// TwinCAT 3 PLC project MC
// ProgramVersion: 3.1.4024.0
// libraries:
//   Tc2_Math, * (Beckhoff Automation GmbH)
//   Tc2_MC2, * (Beckhoff Automation GmbH)
//   Tc2_Standard, * (Beckhoff Automation GmbH)
//   Tc2_System, * (Beckhoff Automation GmbH)
//   Tc2_Utilities, * (Beckhoff Automation GmbH)
//   Tc3_MC2_AdvancedHoming, * (Beckhoff Automation GmbH)
//   Tc3_Module, * (Beckhoff Automation GmbH)
// project tree:
//   GVLs/ motor_settings.TcGVL, robot_settings.TcGVL
//   / PlcTask.TcTTO
//   POUs/Macros/ SYSTIME_MS.TcPOU
//   POUs/MotorInterface/CSP_module/ MotorCSPScheduler.TcPOU
//   POUs/MotorInterface/HM_module/ motor_hm_states_t.TcDUT, MotorHMScheduler.TcPOU
//   POUs/MotorInterface/MotorEnums/ driver_states_t.TcDUT, state_transition_commands_t.TcDUT, driver_modes_t.TcDUT
//   POUs/MotorInterface/MotorIOStructs/ InMotorPDO.TcDUT, OutMotorPDO.TcDUT
//   POUs/MotorInterface/HM_module/temporary_deprecated/ HMConfigIn.TcDUT, HMConfigOut.TcDUT
//   POUs/MotorInterface/ MotorInterface.TcPOU
//   POUs/MotorInterface/PP_module/ MotorPPScheduler.TcPOU, motor_pp_states_t.TcDUT
//   POUs/RobotControl/traj_mode/ RobotTrajScheduler.TcPOU, robot_traj_states_t.TcDUT
//   POUs/RobotControl/hm_mode/ RobotHMScheduler.TcPOU, robot_hm_states_t.TcDUT
//   POUs/RobotControl/pp_mode/ RobotPPScheduler.TcPOU, robot_pp_states_t.TcDUT
//   POUs/RobotControl/RobotKinematics/ InverseKinematics.TcPOU
//   POUs/RobotControl/RobotKinematics/MATH/ ACOSD.TcPOU, ASIND.TcPOU, ATAND.TcPOU, COSD.TcPOU, SIND.TcPOU
//   POUs/RobotControl/ RobotInterface.TcPOU, robot_modes_t.TcDUT
//   VISUs/ MAIN.TcPOU
// real-time tasks:
//   TASK PlcTask: cycle T#1ms, priority 4, ADS port 350
// I/O:
//   DEVICE RobotEtherCAT (disabled), AmsNetId 35.3.62.120.3.1
//     Drive 1 (AZD2A-KED) [AZD2A-KED rev0301]
//   DEVICE Device 3 (EtherCAT), AmsNetId 35.3.234.20.4.1
//     Drive 2 (AZD2A-KED) [AZD2A-KED rev0301]
// variable links:
//   MC/MC Instance <-> Device 3 (EtherCAT)/Drive 2 (AZD2A-KED)
//     PlcTask Inputs/motor_settings.in_motor_pdo[0]/fb_op_mode <-> Axis1 Transmit PDO Mapping 1/Modes of operation display
//     PlcTask Inputs/motor_settings.in_motor_pdo[1]/fb_op_mode <-> Axis2 Transmit PDO Mapping 1/Modes of operation display
//     PlcTask Inputs/motor_settings.in_motor_pdo[0]/fb_position <-> Axis1 Transmit PDO Mapping 1/Position actual value
//     PlcTask Inputs/motor_settings.in_motor_pdo[1]/fb_position <-> Axis2 Transmit PDO Mapping 1/Position actual value
//     PlcTask Inputs/motor_settings.in_motor_pdo[0]/fb_velocity <-> Axis1 Transmit PDO Mapping 1/Velocity actual value
//     PlcTask Inputs/motor_settings.in_motor_pdo[1]/fb_velocity <-> Axis2 Transmit PDO Mapping 1/Velocity actual value
//     PlcTask Inputs/motor_settings.in_motor_pdo[0]/statusword <-> Axis1 Transmit PDO Mapping 1/Statusword
//     PlcTask Inputs/motor_settings.in_motor_pdo[1]/statusword <-> Axis2 Transmit PDO Mapping 1/Statusword
//     PlcTask Outputs/motor_settings.out_motor_pdo[0]/base_current <-> Axis1 Receive PDO Mapping 1/Axis1 base current
//     PlcTask Outputs/motor_settings.out_motor_pdo[1]/base_current <-> Axis2 Receive PDO Mapping 1/Axis2 base current
//     PlcTask Outputs/motor_settings.out_motor_pdo[0]/controlword <-> Axis1 Receive PDO Mapping 1/Controlword
//     PlcTask Outputs/motor_settings.out_motor_pdo[1]/controlword <-> Axis2 Receive PDO Mapping 1/Controlword
//     PlcTask Outputs/motor_settings.out_motor_pdo[0]/motor_op_out <-> Axis1 Receive PDO Mapping 1/Modes of operation
//     PlcTask Outputs/motor_settings.out_motor_pdo[1]/motor_op_out <-> Axis2 Receive PDO Mapping 1/Modes of operation
//     PlcTask Outputs/motor_settings.out_motor_pdo[0]/profile_accel <-> Axis1 Receive PDO Mapping 1/Profile acceleration
//     PlcTask Outputs/motor_settings.out_motor_pdo[1]/profile_accel <-> Axis2 Receive PDO Mapping 1/Profile acceleration
//     PlcTask Outputs/motor_settings.out_motor_pdo[0]/profile_decel <-> Axis1 Receive PDO Mapping 1/Profile deceleration
//     PlcTask Outputs/motor_settings.out_motor_pdo[1]/profile_decel <-> Axis2 Receive PDO Mapping 1/Profile deceleration
//     PlcTask Outputs/motor_settings.out_motor_pdo[0]/profile_vel <-> Axis1 Receive PDO Mapping 1/Profile velocity
//     PlcTask Outputs/motor_settings.out_motor_pdo[1]/profile_vel <-> Axis2 Receive PDO Mapping 1/Profile velocity
//     PlcTask Outputs/motor_settings.out_motor_pdo[0]/target_positon <-> Axis1 Receive PDO Mapping 1/Target position
//     PlcTask Outputs/motor_settings.out_motor_pdo[1]/target_positon <-> Axis2 Receive PDO Mapping 1/Target position
//   MC/MC Instance <-> RobotEtherCAT/Drive 1 (AZD2A-KED)
//     PlcTask Inputs/motor_settings.in_motor_pdo[0]/fb_op_mode <-> Axis1 Transmit PDO Mapping 1/Modes of operation display
//     PlcTask Inputs/motor_settings.in_motor_pdo[1]/fb_op_mode <-> Axis2 Transmit PDO Mapping 1/Modes of operation display
//     PlcTask Inputs/motor_settings.in_motor_pdo[0]/fb_position <-> Axis1 Transmit PDO Mapping 1/Position actual value
//     PlcTask Inputs/motor_settings.in_motor_pdo[1]/fb_position <-> Axis2 Transmit PDO Mapping 1/Position actual value
//     PlcTask Inputs/motor_settings.in_motor_pdo[0]/fb_velocity <-> Axis1 Transmit PDO Mapping 1/Velocity actual value
//     PlcTask Inputs/motor_settings.in_motor_pdo[1]/fb_velocity <-> Axis2 Transmit PDO Mapping 1/Velocity actual value
//     PlcTask Inputs/motor_settings.in_motor_pdo[0]/statusword <-> Axis1 Transmit PDO Mapping 1/Statusword
//     PlcTask Inputs/motor_settings.in_motor_pdo[1]/statusword <-> Axis2 Transmit PDO Mapping 1/Statusword
//     PlcTask Outputs/motor_settings.out_motor_pdo[0]/base_current <-> Axis1 Receive PDO Mapping 1/Axis1 base current
//     PlcTask Outputs/motor_settings.out_motor_pdo[1]/base_current <-> Axis2 Receive PDO Mapping 1/Axis2 base current
//     PlcTask Outputs/motor_settings.out_motor_pdo[0]/controlword <-> Axis1 Receive PDO Mapping 1/Controlword
//     PlcTask Outputs/motor_settings.out_motor_pdo[1]/controlword <-> Axis2 Receive PDO Mapping 1/Controlword
//     PlcTask Outputs/motor_settings.out_motor_pdo[0]/motor_op_out <-> Axis1 Receive PDO Mapping 1/Modes of operation
//     PlcTask Outputs/motor_settings.out_motor_pdo[1]/motor_op_out <-> Axis2 Receive PDO Mapping 1/Modes of operation
//     PlcTask Outputs/motor_settings.out_motor_pdo[0]/profile_accel <-> Axis1 Receive PDO Mapping 1/Profile accel
//     PlcTask Outputs/motor_settings.out_motor_pdo[1]/profile_accel <-> Axis2 Receive PDO Mapping 1/Profile accel
//     PlcTask Outputs/motor_settings.out_motor_pdo[0]/profile_decel <-> Axis1 Receive PDO Mapping 1/Profile decel
//     PlcTask Outputs/motor_settings.out_motor_pdo[1]/profile_decel <-> Axis2 Receive PDO Mapping 1/Profile decel
//     PlcTask Outputs/motor_settings.out_motor_pdo[0]/profile_vel <-> Axis1 Receive PDO Mapping 1/Profile velocity
//     PlcTask Outputs/motor_settings.out_motor_pdo[1]/profile_vel <-> Axis2 Receive PDO Mapping 1/Profile velocity
//     PlcTask Outputs/motor_settings.out_motor_pdo[0]/target_positon <-> Axis1 Receive PDO Mapping 1/Target position
//     PlcTask Outputs/motor_settings.out_motor_pdo[1]/target_positon <-> Axis2 Receive PDO Mapping 1/Target position

CONFIGURATION MC
    RESOURCE PLC ON TwinCAT3
        TASK PlcTask(INTERVAL := T#8ms, PRIORITY := 6);
        PROGRAM MAIN WITH PlcTask : MAIN;
    END_RESOURCE
END_CONFIGURATION

// ---- POUs/MotorInterface/HM_module/motor_hm_states_t.TcDUT
TYPE motor_hm_states_t :
(
	START,
	INPROGRESS,
	END
);
END_TYPE

// ---- POUs/MotorInterface/MotorEnums/driver_states_t.TcDUT
TYPE driver_states_t :
(
	FOO,
	NotReadyToSwitchOn,
	Fault,
	FaultReactionActive,
	SwitchOnDisabled,
	ReadyToSwitchOn,
	SwitchedOn,
	OperationEnabled,
	QuickStopActive
);
END_TYPE

// ---- POUs/MotorInterface/MotorEnums/state_transition_commands_t.TcDUT
TYPE state_transition_commands_t :
(
	Shutdown,
	SwitchOn,
	SwitchOnEnOP,
	DisableVolt,
	QuickStop,
	DisableOP,
	EnableOP,
	FaultReset
);
END_TYPE

// ---- POUs/MotorInterface/MotorIOStructs/InMotorPDO.TcDUT
TYPE InMotorPDO :
STRUCT
	statusword: UINT;
	fb_position: DINT;
	fb_velocity: DINT;
	fb_op_mode: SINT;
END_STRUCT
END_TYPE

// ---- POUs/MotorInterface/MotorIOStructs/OutMotorPDO.TcDUT
TYPE OutMotorPDO :
STRUCT
	controlword: UINT;
	target_positon: DINT;
	motor_op_out: SINT;
	profile_vel: UDINT := 10_000;
	profile_accel: UDINT := 300_000;
	profile_decel: UDINT := 300_000;
	base_current : INT := 1000;
END_STRUCT
END_TYPE

// ---- POUs/MotorInterface/HM_module/temporary_deprecated/HMConfigIn.TcDUT
TYPE HMConfigIn :
STRUCT
	homing_speed: UDINT; // Homing speed, in step/s
	homing_accel: UDINT; // Homing acceleration, in step/s^2
	homing_dir: BOOL;    // Homing direction, true: counter clockwise from top view. false: clockwise from top view.
END_STRUCT
END_TYPE

// ---- POUs/MotorInterface/HM_module/temporary_deprecated/HMConfigOut.TcDUT
TYPE HMConfigOut :
STRUCT
	// For second axis, please add the index offset 0800h. Thus, for axis 2 the index is 6898h, 6899h and 689Ah.
	homing_method: SINT; // Link to the PDO object Homing METHOD (6098h)
	homing_speed: UDINT; // Link to the PDO objects Search speed (6099h.01h/02h)
	homing_accel: UDINT; // Link to the PDO object Homing acceleration (609Ah)
END_STRUCT
END_TYPE

// ---- POUs/MotorInterface/MotorEnums/driver_modes_t.TcDUT
TYPE driver_modes_t :
(
	NI	:=	0,  // Not initiated
	CSP	:=	8,	// Cyclic synchronous position mode
	PP	:=	1,	// Profile position mode
	CSV	:=	9,	// Cyclic synchronous velocity mode
	PV	:=	3,	// Profile velocity mode
	HM	:=	6	// Homing mode
);
END_TYPE

// ---- POUs/MotorInterface/PP_module/motor_pp_states_t.TcDUT
TYPE motor_pp_states_t :
(
	START,
	SENDINGCMD,
	INPROGRESS,
	END
);
END_TYPE

// ---- POUs/RobotControl/traj_mode/robot_traj_states_t.TcDUT
{attribute 'qualified_only'}
{attribute 'strict'}
TYPE robot_traj_states_t :
(
	START,
	RESET,
	READY,
	TRIG,
	EXEC,
	END
);
END_TYPE

// ---- POUs/RobotControl/hm_mode/robot_hm_states_t.TcDUT
{attribute 'qualified_only'}
{attribute 'strict'}
TYPE robot_hm_states_t :
(
	START,
	RETRACT,
	RESETTING_FAULT,
	RELEASE,
	ROTATE,
	HOME,
	END
);
END_TYPE

// ---- POUs/RobotControl/pp_mode/robot_pp_states_t.TcDUT
{attribute 'qualified_only'}
{attribute 'strict'}
TYPE robot_pp_states_t :
(
	START,
	INPROGRESS,
	END
);
END_TYPE

// ---- POUs/RobotControl/robot_modes_t.TcDUT
TYPE robot_modes_t :
( 	HM,
	PP,
	CSP
);
END_TYPE

// ---- GVLs/motor_settings.TcGVL
{attribute 'qualified_only'}
VAR_GLOBAL
	in_motor_pdo		AT%I*: ARRAY[0..1] OF InMotorPDO;
	out_motor_pdo		AT%Q*: ARRAY[0..1] OF OutMotorPDO;	

	motor_interfaces	: ARRAY[0..1] OF MotorInterface[(in_PDO_adr:=ADR(in_motor_pdo[0]),out_PDO_adr:=ADR(out_motor_pdo[0])),
														(in_PDO_adr:=ADR(in_motor_pdo[1]),out_PDO_adr:=ADR(out_motor_pdo[1]))];
	
	pp_scheduler		: ARRAY[0..1] OF MotorPPScheduler[(motor_interface_adr := ADR(motor_interfaces[0])), (motor_interface_adr := ADR(motor_interfaces[1]))];
	csp_scheduler		: ARRAY[0..1] OF MotorCSPScheduler[(motor_interface_adr := ADR(motor_interfaces[0])), (motor_interface_adr := ADR(motor_interfaces[1]))];
	hm_scheduler		: ARRAY[0..1] OF MotorHMScheduler[(motor_interface_adr := ADR(motor_interfaces[0])), (motor_interface_adr := ADR(motor_interfaces[1]))];
END_VAR

// ---- GVLs/robot_settings.TcGVL
{attribute 'qualified_only'}
VAR_GLOBAL
	robot_interface		AT%I*: RobotInterface(	motor_interface_adr:=ADR(motor_settings.motor_interfaces),
											  	pp_scheduler_adr:=ADR(motor_settings.pp_scheduler),
												csp_scheduler_adr:=ADR(motor_settings.csp_scheduler),
												hm_scheduler_adr:=ADR(motor_settings.hm_scheduler));
	// For storing 1_000_000 length trajectories it will take about 8MB. So two trajectories will take no more than 20MB.
	// We applied for a memory that is sufficient for running 1000 sec trajectory.
	// The robot_trajectory_length indicates the indead length of trajectory.
	// Robot trajectory_rotation is the robot's rotation in degree (Not in rad!)
	// Robot's distance is the distance from the center of robot rotor to the center of blade.
	//robot_trajectory_rotation AT%I*: ARRAY[0..1_000_000] OF REAL;
	//robot_trajectory_distance AT%I*: ARRAY[0..1_000_000] OF REAL;
	//robot_trajectory_length AT%I*: UDINT;
	robot_traj_ext : ARRAY [0..1_000_000] OF LREAL;
	robot_traj_rot  : ARRAY [0..1_000_000] OF LREAL;
	// TODO: REMOVE these four temporary variables.
	robot_fb_motor_1 : ARRAY [0..1_000_000] OF LINT;
	robot_fb_motor_2 : ARRAY [0..1_000_000] OF LINT;
	robot_tg_motor_1 : ARRAY [0..1_000_000] OF LINT;
	robot_tg_motor_2 : ARRAY [0..1_000_000] OF LINT;
	
	robot_pp_scheduler		: RobotPPScheduler(robot_interface_adr:=ADR(robot_interface));
	robot_hm_scheduler		: RobotHMScheduler(robot_interface_adr:=ADR(robot_interface));
	robot_traj_scheduler	: RobotTrajScheduler(robot_interface_adr:=ADR(robot_interface),
													robot_trajectory_extension_adr:=ADR(robot_traj_ext),
													robot_trajectory_rotation_adr:=ADR(robot_traj_rot),
													robot_fb_motor_1_adr:=ADR(robot_fb_motor_1),
													robot_fb_motor_2_adr:=ADR(robot_fb_motor_2),
													robot_tg_motor_1_adr:=ADR(robot_tg_motor_1),
													robot_tg_motor_2_adr:=ADR(robot_tg_motor_2));
END_VAR

// ---- VISUs/MAIN.TcPOU
PROGRAM MAIN
VAR
END_VAR

/////////////////////////////////////////////////
///    Update motor data from feedback PDO
/////////////////////////////////////////////////
motor_settings.motor_interfaces[0]();
motor_settings.motor_interfaces[1]();
/////////////////////////////////////////////////
///           Motor Scheduler Loop
/////////////////////////////////////////////////
motor_settings.pp_scheduler[0]();
motor_settings.csp_scheduler[0]();
motor_settings.hm_scheduler[0]();
motor_settings.pp_scheduler[1]();
motor_settings.csp_scheduler[1]();
motor_settings.hm_scheduler[1]();
/////////////////////////////////////////////////
///           Update Robot Interface
/////////////////////////////////////////////////
robot_settings.robot_interface();
robot_settings.robot_pp_scheduler();
robot_settings.robot_hm_scheduler();
robot_settings.robot_traj_scheduler();

END_PROGRAM

// ---- POUs/MotorInterface/MotorInterface.TcPOU
FUNCTION_BLOCK MotorInterface
VAR
	_in_PDO_adr:  POINTER TO InMotorPDO;
	_out_PDO_adr: POINTER TO OutMotorPDO;
		
	_last_position_raw		:	DINT;
	_current_position_raw	:	DINT; 	
	_feedback_position		:	LINT;
	_driver_mode			:	driver_modes_t;
	_driver_state			:	driver_states_t;

	_motor_reset_fault: BOOL;
	
	_switch_threshold:UDINT := 9_000_000;
	_encoder_range: UDINT := 18_000_000;

	_motor_enabled: BOOL;
	_initialized: BOOL := FALSE;
	_last_fault_reset_time : ULINT;
	_motor_reset_fault_flag: BOOL;
	_current_time: ULINT;
END_VAR

(**************Update motor status**************)
_driver_mode:=_in_PDO_adr^.fb_op_mode;
update_position(_in_PDO_adr^.fb_position);
update_statusword(_in_PDO_adr^.statusword);
IF(_motor_enabled) THEN
	(****************Reset fault check****************)
	IF _motor_reset_fault AND (_driver_state = driver_states_t.Fault OR 
		_driver_state = driver_states_t.FaultReactionActive)THEN
		set_driver_operation(state_transition_commands_t.FaultReset);
	END_IF
	(******************Power on motor*****************)
	IF(_driver_state=driver_states_t.NotReadyToSwitchOn) THEN
		set_driver_operation(state_transition_commands_t.Shutdown);
	ELSIF(_driver_state=driver_states_t.SwitchOnDisabled) THEN
		set_driver_operation(state_transition_commands_t.Shutdown);
	ELSIF(_driver_state=driver_states_t.ReadyToSwitchOn) THEN
		set_driver_operation(state_transition_commands_t.SwitchOnEnOP);
	END_IF
ELSE
	set_driver_operation(state_transition_commands_t.DisableVolt);
END_IF
_current_time:=SYSTIME_MS();
IF _motor_reset_fault THEN
	IF NOT _motor_reset_fault_flag THEN
		_motor_reset_fault_flag := TRUE;
		_out_PDO_adr^.controlword.7:=TRUE;
		_last_fault_reset_time := _current_time;
	ELSIF _current_time-_last_fault_reset_time > 500 THEN
		_motor_reset_fault_flag := FALSE;
		_out_PDO_adr^.controlword.7:=FALSE;
	END_IF
END_IF

PROPERTY base_current : INT
GET
base_current := _out_PDO_adr^.base_current;
END_GET
SET
_out_PDO_adr^.base_current:=base_current;
END_SET
END_PROPERTY

PROPERTY controlword_adr : POINTER TO UINT
GET
controlword_adr:=ADR(_out_PDO_adr^.controlword);
END_GET
END_PROPERTY

PROPERTY driver_enable : BOOL
GET
driver_enable:=_motor_enabled;
END_GET
SET
_motor_enabled:=driver_enable;
END_SET
END_PROPERTY

PROPERTY driver_mode : driver_modes_t
GET
driver_mode:=_driver_mode;
END_GET
SET
_out_PDO_adr^.motor_op_out:=TO_SINT(driver_mode);
END_SET
END_PROPERTY

PROPERTY driver_state : driver_states_t
GET
driver_state:=_driver_state;
END_GET
END_PROPERTY

PROPERTY encoder_range : UDINT
GET
encoder_range:=_encoder_range;
END_GET
SET
_encoder_range:=encoder_range;
_switch_threshold:=TO_UDINT(_encoder_range/2);
END_SET
END_PROPERTY

METHOD FB_init : BOOL
VAR_INPUT
	bInitRetains : BOOL; // if TRUE, the retain variables are initialized (warm start / cold start)
	bInCopyCode : BOOL;  // if TRUE, the instance afterwards gets moved into the copy code (online change)
	in_PDO_adr : POINTER TO InMotorPDO;
	out_PDO_adr : POINTER TO OutMotorPDO;
END_VAR
_in_PDO_adr:=in_PDO_adr;
_out_PDO_adr:=out_PDO_adr;
END_METHOD

{attribute 'qualified_only'}
PROPERTY feedback_position : LINT
GET
{attribute 'qualified_only'}
VAR
END_VAR
feedback_position:=_feedback_position;
END_GET
END_PROPERTY

PROPERTY raw_position : DINT
GET
raw_position:=_current_position_raw;
END_GET
END_PROPERTY

PROPERTY reset_fault : BOOL
GET
reset_fault:=_motor_reset_fault;
END_GET
SET
_motor_reset_fault:=reset_fault;
END_SET
END_PROPERTY

METHOD reset_position : BOOL
VAR_INPUT
END_VAR
_feedback_position:=0;
END_METHOD

METHOD PRIVATE set_driver_operation : BOOL
VAR_INPUT
	state_transition_command: state_transition_commands_t;
END_VAR
CASE state_transition_command OF
	Shutdown: _out_PDO_adr^.controlword:=16#06;
	SwitchOn: _out_PDO_adr^.controlword:=16#07;
	SwitchOnEnOP: _out_PDO_adr^.controlword:=16#0F;
	DisableVolt: _out_PDO_adr^.controlword:=16#00;
	QuickStop: _out_PDO_adr^.controlword:=16#02;
	DisableOP: _out_PDO_adr^.controlword:=16#07;
	EnableOP: _out_PDO_adr^.controlword:=16#0F;
	FaultReset: _out_PDO_adr^.controlword:=16#80;
END_CASE
END_METHOD

METHOD set_PP_parameters : BOOL
VAR_INPUT
	profile_velocity : UDINT;
	profile_acceleration: UDINT;
END_VAR
_out_PDO_adr^.profile_vel:=profile_velocity;
_out_PDO_adr^.profile_accel:=profile_acceleration;
_out_PDO_adr^.profile_decel:=profile_acceleration;
END_METHOD

PROPERTY statusword : UINT
GET
statusword:=_in_PDO_adr^.statusword;
END_GET
END_PROPERTY

PROPERTY target_position : DINT
GET
target_position:=_out_PDO_adr^.target_positon;
END_GET
SET
_out_PDO_adr^.target_positon:=target_position;
END_SET
END_PROPERTY

METHOD PRIVATE update_position : BOOL
(**********Update Position**********
@brief:	Update the position of motor from the signal from motor. Since the
		encoder has limited value range, when the value exceeding the maxi-
		mum value, it will jumps to the minimum value. This method will un-
		wrap the value to ensure the feedback position is continuous.
@param:	statusword	[in] The DINT value from motor PDO.
					which the EtherCAT index should be 0x6064:00, 0x6864:00
*)
VAR_INPUT
	motor_position_raw: DINT;
END_VAR
VAR
	angle_offset: DINT;
END_VAR
IF(NOT _initialized) THEN
	_last_position_raw := motor_position_raw;
	_feedback_position := motor_position_raw;
	_initialized := TRUE;
END_IF
_current_position_raw := motor_position_raw;
angle_offset := _current_position_raw - _last_position_raw;
IF (ABS(angle_offset) > _switch_threshold) THEN
	angle_offset := angle_offset - angle_offset/ABS(angle_offset)*_encoder_range;
END_IF
_feedback_position := _feedback_position+angle_offset;
_last_position_raw := _current_position_raw;
END_METHOD

METHOD update_rounds : BOOL
VAR_INPUT
	round_count : DINT;
END_VAR
_feedback_position := _feedback_position + round_count * _encoder_range;
END_METHOD

METHOD PRIVATE update_statusword
(**********Update Statusword**********
@brief:	Translate statuswords to motor driver states,
		the translated statuswords is stored in the 
		driver_state variable.
@param:	statusword	[in] The UINT value from motor PDO.
					which the EtherCAT index should be 0x6041:00, 0x6841:00
*)
VAR_INPUT
	statusword: UINT;
END_VAR
VAR
	status_bits: USINT;
END_VAR
(*State process part*)
// The bit 0-6 of statusword indicates the status output.
// To get the status state, we first shift one bit left,
// then crop and finally shift the bit back. 
// 1. xxxx xxxx xxxx xxxx           ->           2. xxxx xxxx xxxx xxx0 ->
//               |------|   left shift 1 bit                 |  Crop  |  
//             What we want                                  with SINT
// 3. xxxx xxx0                     ->           4. 0xxx xxxx
//   Cropped data          right shift one bit       Result
status_bits := SHR(TO_USINT(SHL(statusword,1)),1);
// Switch case for the status output, refer to AZD user manual pp.55.
CASE status_bits OF
	16#00:			_driver_state:=driver_states_t.NotReadyToSwitchOn;
	16#28,16#38:	_driver_state:=driver_states_t.Fault;
	16#2F,16#3F:	_driver_state:=driver_states_t.FaultReactionActive;
	16#60,16#70:	_driver_state:=driver_states_t.SwitchOnDisabled;
	16#21,16#31:	_driver_state:=driver_states_t.ReadyToSwitchOn;
	16#23,16#33:	_driver_state:=driver_states_t.SwitchedOn;
	16#27,16#37:	_driver_state:=driver_states_t.OperationEnabled;
	16#07,16#17:	_driver_state:=driver_states_t.QuickStopActive;
ELSE
	_driver_state := driver_states_t.FOO;
END_CASE
END_METHOD

END_FUNCTION_BLOCK

// ---- POUs/Macros/SYSTIME_MS.TcPOU
FUNCTION SYSTIME_MS : ULINT
VAR_INPUT
END_VAR
VAR
	time_low_dw: UDINT;
	time_upper_dw:UDINT;
	curr_time:ULINT;
	systime:GETSYSTEMTIME;
	curr_time_raw: ULINT;
END_VAR

systime(timeLoDW=>time_low_dw, timeHiDW=>time_upper_dw);
(*curr_time := time_upper_dw;
curr_time := SHL(curr_time,32)+time_low_dw;
// Curr time has a unit of 100ns. We need to convert it to ms by divide it with 10,000.
SYSTIME_MS := REAL_TO_ULINT(TO_REAL(curr_time)/10_000);  *)
SYSTIME_MS := LREAL_TO_ULINT(TO_LREAL(F_GetSystemTime()/10_000));

END_FUNCTION

// ---- POUs/MotorInterface/PP_module/MotorPPScheduler.TcPOU
FUNCTION_BLOCK MotorPPScheduler
VAR
	_skd_state: motor_pp_states_t:=motor_pp_states_t.END;
	_profile_velocity: UDINT:= 10000;
	_profile_acceleration: UDINT:= 300000;
	
	_change_immediately: BOOL;
	_reference_coordinate: BOOL;
	_push_operation: BOOL;
	
	_target_position: DINT;
	_motor_interface_adr: POINTER TO MotorInterface;
	
	_statusword: UINT;
	_controlword_adr : POINTER TO UINT;
	_last_send_time: ULINT;
	_MSG_SENT:BOOL:=FALSE;
END_VAR

IF _motor_interface_adr^.driver_mode=driver_modes_t.PP AND _motor_interface_adr^.driver_enable AND _motor_interface_adr^.driver_state<>driver_states_t.Fault AND _motor_interface_adr^.driver_state<>driver_states_t.FaultReactionActive THEN
	_statusword := _motor_interface_adr^.statusword;
	_motor_interface_adr^.set_PP_parameters(profile_velocity:=_profile_velocity, profile_acceleration:=_profile_acceleration);
	_controlword_adr^.5:=_change_immediately;
	_controlword_adr^.6:=_reference_coordinate;
	_controlword_adr^.13:=_push_operation;
	
	CASE _skd_state OF
		motor_pp_states_t.START: 
			_skd_state:=motor_pp_states_t.SENDINGCMD;
			_controlword_adr^.4:=0;
			_MSG_SENT:=FALSE;
		motor_pp_states_t.SENDINGCMD:
			_controlword_adr^.4:=1;
			IF NOT _MSG_SENT THEN
				_last_send_time:=SYSTIME_MS();
			END_IF
			_MSG_SENT:=TRUE;
			IF _statusword.12 THEN
				_skd_state := motor_pp_states_t.INPROGRESS;
			ELSIF (SYSTIME_MS()-_last_send_time)>500 THEN
				_MSG_SENT:=FALSE;
				_controlword_adr^.4:=0;
			END_IF
		motor_pp_states_t.INPROGRESS:
			_controlword_adr^.4:=1;
			// 10 is end to target, while 15 is reaches to torque limit (limited by mechanical structure)
			IF _statusword.10 OR _statusword.15 THEN
				_skd_state := motor_pp_states_t.END;
			END_IF
		motor_pp_states_t.END:
			_controlword_adr^.4:=0;
	END_CASE
	_motor_interface_adr^.target_position:=_target_position;
END_IF

METHOD activate : BOOL
VAR_INPUT
END_VAR
_motor_interface_adr^.driver_mode:=driver_modes_t.PP;
END_METHOD

METHOD FB_init : BOOL
VAR_INPUT
	bInitRetains : BOOL; // if TRUE, the retain variables are initialized (warm start / cold start)
	bInCopyCode : BOOL;  // if TRUE, the instance afterwards gets moved into the copy code (online change)
	motor_interface_adr : POINTER TO MotorInterface;
END_VAR
_motor_interface_adr := motor_interface_adr;
_controlword_adr := _motor_interface_adr^.controlword_adr;
END_METHOD

{attribute 'TcRpcEnable'}
METHOD get_state : motor_pp_states_t
VAR_INPUT
END_VAR
get_state:=_skd_state;
END_METHOD

{attribute 'TcRpcEnable'}
METHOD start_operation : BOOL
VAR_INPUT
	target_position: LINT;
	change_immediately: BOOL;
	reference_coordinate: BOOL;
	push_operation: BOOL;
END_VAR
_change_immediately:=change_immediately;
_reference_coordinate:=reference_coordinate;
_push_operation:=push_operation;
IF(reference_coordinate) THEN
	_target_position := TO_DINT(target_position);
ELSE
	_target_position := TO_DINT(target_position - _motor_interface_adr^.feedback_position + _motor_interface_adr^.raw_position);
END_IF
_skd_state:=motor_pp_states_t.START;
END_METHOD

METHOD update_pp_parameter : BOOL
VAR_INPUT
	profile_velocity:UDINT;
	profile_acceleration:UDINT;
END_VAR
_profile_velocity:=profile_velocity;
_profile_acceleration:=profile_acceleration;
END_METHOD

END_FUNCTION_BLOCK

// ---- POUs/MotorInterface/CSP_module/MotorCSPScheduler.TcPOU
FUNCTION_BLOCK MotorCSPScheduler
VAR
	_target_position:LINT;
	_motor_interface_adr: POINTER TO MotorInterface;
	_controlword_adr : POINTER TO UINT;
END_VAR

IF _motor_interface_adr^.driver_mode = driver_modes_t.CSP AND _motor_interface_adr^.driver_enable THEN
	_motor_interface_adr^.target_position := TO_DINT(_target_position - 
								MODTURNS(	_motor_interface_adr^._feedback_position,
											_motor_interface_adr^.encoder_range)*
											TO_LINT(_motor_interface_adr^.encoder_range));
	_controlword_adr^.4:=TRUE;
END_IF

METHOD activate : BOOL
VAR_INPUT
	
END_VAR
_motor_interface_adr^.driver_mode:=driver_modes_t.CSP;
END_METHOD

METHOD FB_init : BOOL
VAR_INPUT
	bInitRetains : BOOL; // if TRUE, the retain variables are initialized (warm start / cold start)
	bInCopyCode : BOOL;  // if TRUE, the instance afterwards gets moved into the copy code (online change)
	motor_interface_adr: POINTER TO MotorInterface;
END_VAR
_motor_interface_adr := motor_interface_adr;
_controlword_adr:=_motor_interface_adr^.controlword_adr;
END_METHOD

{attribute 'TcRpcEnable'}
METHOD set_position : BOOL
VAR_INPUT
	target_position: LINT;
END_VAR
_target_position := target_position;
END_METHOD

END_FUNCTION_BLOCK

// ---- POUs/MotorInterface/HM_module/MotorHMScheduler.TcPOU
FUNCTION_BLOCK MotorHMScheduler
VAR
	_motor_interface_adr: POINTER TO MotorInterface;
	_operation_start_time : ULINT;
	_skd_state : motor_hm_states_t:=motor_hm_states_t.END;
	
	_statusword: UINT;
	_controlword_adr : POINTER TO UINT;
END_VAR

IF _motor_interface_adr^.driver_mode=driver_modes_t.HM AND _motor_interface_adr^.driver_enable THEN
	_statusword:=_motor_interface_adr^.statusword;
	CASE _skd_state OF
		motor_hm_states_t.START:
			_controlword_adr^.4:=0;
			_skd_state := motor_hm_states_t.INPROGRESS;
			_operation_start_time := SYSTIME_MS(); 
		motor_hm_states_t.INPROGRESS:
			_controlword_adr^.4:=1;
			IF(_statusword.10 AND _statusword.12) THEN
				_skd_state := motor_hm_states_t.END;
			END_IF
		motor_hm_states_t.END:
			_controlword_adr^.4:=0;
	END_CASE
END_IF

METHOD activate : BOOL
VAR_INPUT
END_VAR
_motor_interface_adr^.driver_mode:=driver_modes_t.HM;
END_METHOD

METHOD FB_init : BOOL
VAR_INPUT
	bInitRetains : BOOL; // if TRUE, the retain variables are initialized (warm start / cold start)
	bInCopyCode : BOOL;  // if TRUE, the instance afterwards gets moved into the copy code (online change)
	motor_interface_adr : POINTER TO MotorInterface;
END_VAR
_motor_interface_adr := motor_interface_adr;
_controlword_adr:=_motor_interface_adr^.controlword_adr;
END_METHOD

METHOD get_state : motor_hm_states_t
VAR_INPUT
END_VAR
get_state:=_skd_state;
END_METHOD

{attribute 'TcRpcEnable'}
METHOD start_operation : BOOL
VAR_INPUT
END_VAR
_skd_state := motor_hm_states_t.START;
END_METHOD

END_FUNCTION_BLOCK

// ---- POUs/RobotControl/RobotInterface.TcPOU
FUNCTION_BLOCK RobotInterface
VAR_INPUT
END_VAR
VAR_OUTPUT
	
END_VAR
VAR
	_initialized : BOOL := FALSE;
	_robot_enabled : BOOL:= FALSE;
	_robot_reset_fault: BOOL:=FALSE;
	_robot_mode : robot_modes_t := robot_modes_t.PP;
	_motor_interface_adr: POINTER TO ARRAY[0..1] OF MotorInterface;
	_motor_pp_scheduler_adr: POINTER TO ARRAY[0..1] OF MotorPPScheduler;
	_motor_csp_scheduler_adr: POINTER TO ARRAY[0..1] OF MotorCSPScheduler;
	_motor_hm_scheduler_adr: POINTER TO ARRAY[0..1] OF MotorHMScheduler;
	_ud_rounds:DINT;
END_VAR
VAR_IN_OUT
END_VAR

IF (NOT _initialized) AND 	_motor_interface_adr^[0].driver_state<>driver_states_t.Fault AND _motor_interface_adr^[0].driver_state<>driver_states_t.FaultReactionActive AND
							_motor_interface_adr^[1].driver_state<>driver_states_t.Fault AND _motor_interface_adr^[1].driver_state<>driver_states_t.FaultReactionActive THEN
	// Start angle calibration. If the motor angles is near the upper/lower bound of encoder, 
	// there might have values like: feedback_angle[0] = -8_999_999, feedback_angle[1] = 8_999_999. In this case, we need to wrap motor angles
	// to feedback_angle[0] = 9_000_001. To judge if it happened, we simply compare the robot's feedback positions. If the positions are larger
	// than 1 round (1_000_000 steps), we can determine that this occasion happens, since robot's mechanical structure limits the two motor's 
	// angle difference in 1 round.
	IF ABS(	_motor_interface_adr^[0].feedback_position - _motor_interface_adr^[1].feedback_position) > 1_000_000 THEN
			_motor_interface_adr^[0].update_rounds(TO_DINT(_motor_interface_adr^[0].feedback_position < _motor_interface_adr^[1].feedback_position)*2-1);
	END_IF
	_ud_rounds:=TO_DINT(_motor_interface_adr^[0].feedback_position < _motor_interface_adr^[1].feedback_position)*2-1;
	_initialized := TRUE;
END_IF
IF _robot_enabled THEN
	_motor_interface_adr^[0].driver_enable:=TRUE;
	_motor_interface_adr^[1].driver_enable:=TRUE;
END_IF
IF _robot_reset_fault THEN
	IF 	_motor_interface_adr^[0].driver_state=driver_states_t.Fault OR _motor_interface_adr^[0].driver_state=driver_states_t.FaultReactionActive THEN
		_motor_interface_adr^[0].reset_fault:=TRUE;
	END_IF
	IF	_motor_interface_adr^[1].driver_state=driver_states_t.Fault OR _motor_interface_adr^[1].driver_state=driver_states_t.FaultReactionActive THEN
		_motor_interface_adr^[1].reset_fault:=TRUE;
	END_IF
	IF 	_motor_interface_adr^[0].driver_state<>driver_states_t.Fault AND _motor_interface_adr^[0].driver_state<>driver_states_t.FaultReactionActive AND
		_motor_interface_adr^[1].driver_state<>driver_states_t.Fault AND _motor_interface_adr^[1].driver_state<>driver_states_t.FaultReactionActive THEN
		_robot_reset_fault:=FALSE;
		_motor_interface_adr^[0].reset_fault:=FALSE;
		_motor_interface_adr^[1].reset_fault:=FALSE;
	END_IF
END_IF

METHOD FB_init : BOOL
VAR_INPUT
	bInitRetains : BOOL; // if TRUE, the retain variables are initialized (warm start / cold start)
	bInCopyCode : BOOL;  // if TRUE, the instance afterwards gets moved into the copy code (online change)
	motor_interface_adr: POINTER TO ARRAY[0..1] OF MotorInterface;
	csp_scheduler_adr: POINTER TO ARRAY[0..1] OF MotorCSPScheduler;
	pp_scheduler_adr: POINTER TO ARRAY[0..1] OF MotorPPScheduler;
	hm_scheduler_adr: POINTER TO ARRAY[0..1] OF MotorHMScheduler;
END_VAR
_motor_interface_adr := motor_interface_adr;
_motor_pp_scheduler_adr:=pp_scheduler_adr;
_motor_csp_scheduler_adr:=csp_scheduler_adr;
_motor_hm_scheduler_adr:=hm_scheduler_adr;
END_METHOD

PROPERTY motor_csp_scheduler_adr : POINTER TO ARRAY[0..1] OF MotorCSPScheduler
GET
motor_csp_scheduler_adr := _motor_csp_scheduler_adr;
END_GET
END_PROPERTY

PROPERTY motor_hm_scheduler_adr : POINTER TO ARRAY[0..1] OF MotorHMScheduler
GET
motor_hm_scheduler_adr := _motor_hm_scheduler_adr;
END_GET
END_PROPERTY

PROPERTY motor_interface_adr : POINTER TO ARRAY[0..1] OF MotorInterface
GET
motor_interface_adr:=_motor_interface_adr;
END_GET
END_PROPERTY

PROPERTY motor_pp_scheduler_adr : POINTER TO ARRAY[0..1] OF MotorPPScheduler
GET
motor_pp_scheduler_adr := _motor_pp_scheduler_adr;
END_GET
END_PROPERTY

{attribute 'TcRpcEnable'}
PROPERTY robot_enabled : BOOL
GET
robot_enabled:=_robot_enabled;
END_GET
SET
_robot_enabled:=robot_enabled;
END_SET
END_PROPERTY

PROPERTY robot_mode : robot_modes_t
GET
robot_mode:=_robot_mode;
END_GET
SET
_robot_mode:=robot_mode;
END_SET
END_PROPERTY

{attribute 'TcRpcEnable'}
PROPERTY robot_reset_fault : BOOL
GET
robot_reset_fault:=_robot_reset_fault;
END_GET
SET
_robot_reset_fault:=robot_reset_fault;
END_SET
END_PROPERTY

END_FUNCTION_BLOCK

// ---- POUs/RobotControl/pp_mode/RobotPPScheduler.TcPOU
FUNCTION_BLOCK RobotPPScheduler
VAR
	/// Interfaces
	_robot_interface_adr: POINTER TO RobotInterface;
	_motor_pp_scheduler_adr: POINTER TO ARRAY[0..1] OF MotorPPScheduler;
END_VAR
VAR
	/// Runtime variables
	_robot_state : robot_pp_states_t:=robot_pp_states_t.END;
	_target_distance: LREAL;
	_target_angle : LREAL;
	_motor_angles : ARRAY[0..1] OF DINT;
END_VAR

IF(_robot_interface_adr^.robot_mode=robot_modes_t.PP  AND _robot_interface_adr^.robot_enabled) THEN
	CASE _robot_state OF
		robot_pp_states_t.START:
			_motor_pp_scheduler_adr^[0].activate();
			_motor_pp_scheduler_adr^[1].activate();
			InverseKinematics(	target_dist:=_target_distance, 
								target_angle:=_target_angle,
								motor_axis1_angle=>_motor_angles[0],
								motor_axis2_angle=>_motor_angles[1]);
			_motor_pp_scheduler_adr^[0].start_operation(
									target_position:=_motor_angles[0],
									change_immediately:=TRUE,
									reference_coordinate:=FALSE,
									push_operation:=FALSE);
			_motor_pp_scheduler_adr^[1].start_operation(
									target_position:=_motor_angles[1],
									change_immediately:=TRUE,
									reference_coordinate:=FALSE,
									push_operation:=FALSE);
			_robot_state:=robot_pp_states_t.INPROGRESS;
		robot_pp_states_t.INPROGRESS:
			IF(_motor_pp_scheduler_adr^[0].get_state()=motor_pp_states_t.END AND _motor_pp_scheduler_adr^[1].get_state()=motor_pp_states_t.END) THEN
				_robot_state:=robot_pp_states_t.END;
			END_IF
	END_CASE
END_IF

{attribute 'TcRpcEnable'}
METHOD activate : BOOL
VAR_INPUT
END_VAR

_robot_interface_adr^.robot_mode:=robot_modes_t.PP;
_robot_state:=robot_pp_states_t.END;
END_METHOD

METHOD FB_init : BOOL
VAR_INPUT
	bInitRetains : BOOL; // if TRUE, the retain variables are initialized (warm start / cold start)
	bInCopyCode : BOOL;  // if TRUE, the instance afterwards gets moved into the copy code (online change)
	robot_interface_adr: POINTER TO RobotInterface;
END_VAR
_robot_interface_adr:=robot_interface_adr;
_motor_pp_scheduler_adr:=_robot_interface_adr^.motor_pp_scheduler_adr;
END_METHOD

{attribute 'TcRpcEnable'}
METHOD get_state : robot_pp_states_t
VAR_INPUT
END_VAR
get_state:=_robot_state;
END_METHOD

{attribute 'TcRpcEnable'}
METHOD start_operation : BOOL
VAR_INPUT
	target_distance: LREAL;
	target_angle : LREAL;
END_VAR
_robot_interface_adr^.robot_enabled:=TRUE;
_target_distance:=target_distance;
_target_angle:=target_angle;
_robot_state:=robot_pp_states_t.START;
END_METHOD

END_FUNCTION_BLOCK

// ---- POUs/RobotControl/RobotKinematics/InverseKinematics.TcPOU
FUNCTION InverseKinematics
VAR_INPUT
	target_dist: LREAL;
	target_angle: LREAL;
END_VAR
VAR_OUTPUT
	motor_axis1_angle: DINT;
	motor_axis2_angle: DINT;
END_VAR
VAR
	(*pre-loaded parameters for calculate robot dimensions*)
	(*Solve link lenghts analytically. 
		Preloaded parameter so only perform calculation once, at program initialization.*)
	// l2: Blade joint distance
	l2:LREAL := 50.84/2;
	// l3: Front arm
	l3:LREAL := 217;
	x41:LREAL:= 102*COSD(45);
	y41:LREAL:= 102*SIND(45);
	x42:LREAL:= 100/SIND(43)*COSD(2);
	y42:LREAL:= 100/SIND(43)*SIND(2);
	x4s:LREAL:= x41+x42;
	y4s:LREAL:= y41+y42;
	// l4: Rear arm
	l4:LREAL:=SQRT(EXPT(x4s,2)+EXPT(y4s,2));
	
	// The arm's angle from home position, see documentation. 
	home_angle_deg:LREAL:=81.5+ATAND(y4s/x4s);
	a3_rad:LREAL:=ACOS((l4*SIND(home_angle_deg)-l2)/l3);
	center_offset:LREAL:=l3*SIN(a3_rad)-l4*COSD(180-home_angle_deg);
	// l1: Blade length, from joint to center position, range from 173 mm to 606.5 mm.
	l1:LREAL:=199.5-center_offset;
	
	(*Inverse kinematic calculation variables*)
	angle1_deg:LREAL;
	angle2_deg:LREAL;
	arm_rot_offset_deg:LREAL;
END_VAR

// Crop target dist in operation range.
IF target_dist < 173 THEN
	target_dist:= 173;
ELSIF target_dist > 630 THEN
	target_dist:= 630;
END_IF

angle1_deg:=ATAND(l2/(target_dist-l1));
angle2_deg:=ACOSD((EXPT(target_dist-l1,2)+EXPT(l2,2)+EXPT(l4,2)-EXPT(l3,2))
			/(2*SQRT(EXPT(target_dist-l1,2)+EXPT(l2,2))*l4));
arm_rot_offset_deg:=angle1_deg+angle2_deg-home_angle_deg;

motor_axis1_angle:= TO_DINT((target_angle+arm_rot_offset_deg)/360*1_000_000);
motor_axis2_angle:= TO_DINT((target_angle-arm_rot_offset_deg)/360*1_000_000);

END_FUNCTION

// ---- POUs/RobotControl/RobotKinematics/MATH/COSD.TcPOU
FUNCTION COSD : LREAL
VAR_INPUT
	ANGLE:LREAL;
END_VAR
VAR
END_VAR

COSD:=COS(DEG_TO_RAD(ANGLE));

END_FUNCTION

// ---- POUs/RobotControl/RobotKinematics/MATH/SIND.TcPOU
FUNCTION SIND : LREAL
VAR_INPUT
	ANGLE:LREAL;
END_VAR
VAR
END_VAR

SIND:=SIN(DEG_TO_RAD(ANGLE));

END_FUNCTION

// ---- POUs/RobotControl/RobotKinematics/MATH/ATAND.TcPOU
FUNCTION ATAND : LREAL
VAR_INPUT
	TANVAL: LREAL;
END_VAR
VAR
END_VAR

ATAND:=RAD_TO_DEG(ATAN(TANVAL));

END_FUNCTION

// ---- POUs/RobotControl/RobotKinematics/MATH/ACOSD.TcPOU
FUNCTION ACOSD : LREAL
VAR_INPUT
	COSVAL:LREAL;
END_VAR
VAR
END_VAR

ACOSD:=RAD_TO_DEG(ACOS(COSVAL));

END_FUNCTION

// ---- POUs/RobotControl/hm_mode/RobotHMScheduler.TcPOU
FUNCTION_BLOCK RobotHMScheduler
VAR_OUTPUT
END_VAR
VAR
	_robot_state : robot_hm_states_t:=robot_hm_states_t.END;
	_robot_direction: LINT;
	_rotation_angle: LINT;
	
	_robot_interface_adr: POINTER TO RobotInterface;
	_motor_interface_adr: POINTER TO ARRAY[0..1] OF MotorInterface;
	_motor_pp_scheduler_adr: POINTER TO ARRAY[0..1] OF MotorPPScheduler;
	_motor_hm_scheduler_adr: POINTER TO ARRAY[0..1] OF MotorHMScheduler;
	_motor_csp_scheduler_adr: POINTER TO ARRAY[0..1] OF MotorCSPScheduler;
END_VAR

IF(_robot_interface_adr^.robot_mode=robot_modes_t.HM AND _robot_interface_adr^.robot_enabled) THEN
CASE _robot_state OF
	robot_hm_states_t.START:
		_motor_interface_adr^[0].driver_enable:=TRUE;
		_motor_interface_adr^[1].driver_enable:=TRUE;
		_motor_interface_adr^[0].base_current:=70;
		_motor_interface_adr^[1].base_current:=70;
		_motor_pp_scheduler_adr^[0].update_pp_parameter(profile_velocity:=30000,profile_acceleration:=5000);
		_motor_pp_scheduler_adr^[1].update_pp_parameter(profile_velocity:=30000,profile_acceleration:=5000);
		_motor_pp_scheduler_adr^[0].activate();
		_motor_pp_scheduler_adr^[1].activate();
		_motor_pp_scheduler_adr^[0].start_operation(target_position:=500_000, change_immediately:=FALSE,reference_coordinate:=TRUE,push_operation:=FALSE);
		_motor_pp_scheduler_adr^[1].start_operation(target_position:=-500_000, change_immediately:=FALSE,reference_coordinate:=TRUE,push_operation:=FALSE);
		_robot_interface_adr^.robot_reset_fault:=FALSE;
		_robot_state := robot_hm_states_t.RETRACT;
	robot_hm_states_t.RETRACT:
		IF(	(_motor_interface_adr^[0].driver_state=driver_states_t.Fault OR _motor_interface_adr^[0].driver_state=driver_states_t.FaultReactionActive) AND
			(_motor_interface_adr^[1].driver_state=driver_states_t.Fault OR _motor_interface_adr^[1].driver_state=driver_states_t.FaultReactionActive)) THEN
			_robot_interface_adr^.robot_reset_fault:=TRUE;
			_robot_state := robot_hm_states_t.RESETTING_FAULT;
		END_IF
	robot_hm_states_t.RESETTING_FAULT:
		IF(	_motor_interface_adr^[0].driver_state<>driver_states_t.Fault AND _motor_interface_adr^[0].driver_State<>driver_states_t.FaultReactionActive AND
			_motor_interface_adr^[1].driver_state<>driver_states_t.Fault AND _motor_interface_adr^[1].driver_state<>driver_states_t.FaultReactionActive) THEN
			_robot_interface_adr^.robot_reset_fault:=FALSE;
			_motor_interface_adr^[0].base_current:=1000;
			_motor_interface_adr^[1].base_current:=1000;
			_motor_pp_scheduler_adr^[0].start_operation(target_position:=-20000, change_immediately:=TRUE,reference_coordinate:=TRUE,push_operation:=FALSE);
			_motor_pp_scheduler_adr^[1].start_operation(target_position:=20000, change_immediately:=TRUE,reference_coordinate:=TRUE,push_operation:=FALSE);
			_robot_state := robot_hm_states_t.RELEASE;
		END_IF
	robot_hm_states_t.RELEASE:
		IF(_motor_pp_scheduler_adr^[0].get_state()=motor_pp_states_t.END AND _motor_pp_scheduler_adr^[1].get_state()=motor_pp_states_t.END) THEN
			_robot_direction:= TO_LINT(_motor_interface_adr^[0].feedback_position + _motor_interface_adr^[1].feedback_position)/2;
			_rotation_angle:=LREAL_TO_LINT(TO_LREAL(_robot_direction)/1_000_000)*1_000_000 - _robot_direction;
			_motor_pp_scheduler_adr^[0].start_operation(target_position:=_rotation_angle, change_immediately:=TRUE,reference_coordinate:=TRUE,push_operation:=FALSE);
			_motor_pp_scheduler_adr^[1].start_operation(target_position:=_rotation_angle, change_immediately:=TRUE,reference_coordinate:=TRUE,push_operation:=FALSE);
			_robot_state := robot_hm_states_t.ROTATE;
		END_IF
	robot_hm_states_t.ROTATE:
		IF(_motor_pp_scheduler_adr^[0].get_state()=motor_pp_states_t.END AND _motor_pp_scheduler_adr^[1].get_state()=motor_pp_states_t.END) THEN
			_motor_hm_scheduler_adr^[0].activate();
			_motor_hm_scheduler_adr^[1].activate();
			_motor_hm_scheduler_adr^[0].start_operation();
			_motor_hm_scheduler_adr^[1].start_operation();
			_robot_state := robot_hm_states_t.HOME;
		END_IF
	robot_hm_states_t.HOME:
		IF(_motor_hm_scheduler_adr^[0].get_state() = motor_hm_states_t.END AND _motor_hm_scheduler_adr^[1].get_state()=motor_hm_states_t.END) THEN
			_robot_state := robot_hm_states_t.END;
			_motor_interface_adr^[0].reset_position();
			_motor_interface_adr^[1].reset_position();
		END_IF
END_CASE
END_IF

{attribute 'TcRpcEnable'}
METHOD activate : BOOL
VAR_INPUT
END_VAR
_robot_interface_adr^.robot_mode:=robot_modes_t.HM;
_robot_state:=robot_hm_states_t.END;
END_METHOD

METHOD FB_init : BOOL
VAR_INPUT
	bInitRetains : BOOL; // if TRUE, the retain variables are initialized (warm start / cold start)
	bInCopyCode : BOOL;  // if TRUE, the instance afterwards gets moved into the copy code (online change)
	robot_interface_adr: POINTER TO RobotInterface;
END_VAR
_robot_interface_adr:=robot_interface_adr;
_motor_pp_scheduler_adr:=robot_interface_adr^.motor_pp_scheduler_adr;
_motor_hm_scheduler_adr:=robot_interface_adr^.motor_hm_scheduler_adr;
_motor_csp_scheduler_adr:=robot_interface_adr^.motor_csp_scheduler_adr;
_motor_interface_adr:=robot_interface_adr^.motor_interface_adr;
END_METHOD

{attribute 'TcRpcEnable'}
METHOD get_state : robot_hm_states_t
VAR_INPUT
END_VAR
get_state:=_robot_state;
END_METHOD

{attribute 'TcRpcEnable'}
METHOD start_operation : BOOL
VAR_INPUT
END_VAR
_robot_interface_adr^.robot_enabled:=TRUE;
_robot_state := robot_hm_states_t.START;
END_METHOD

END_FUNCTION_BLOCK

// ---- POUs/RobotControl/traj_mode/RobotTrajScheduler.TcPOU
FUNCTION_BLOCK RobotTrajScheduler
VAR_INPUT
END_VAR
VAR_OUTPUT
END_VAR
VAR
	_robot_interface_adr: POINTER TO RobotInterface;
	_motor_interface_adr: POINTER TO ARRAY[0..1] OF MotorInterface;
	_motor_pp_scheduler_adr: POINTER TO ARRAY[0..1] OF MotorPPScheduler;
	_motor_hm_scheduler_adr: POINTER TO ARRAY[0..1] OF MotorHMScheduler;
	_motor_csp_scheduler_adr: POINTER TO ARRAY[0..1] OF MotorCSPScheduler;
	
	_target_motor_angles : ARRAY[0..1] OF DINT;
	_robot_state: robot_traj_states_t :=robot_traj_states_t.END;
	_robot_trajectory_extension_adr : POINTER TO ARRAY [0..1000000] OF LREAL;
	_robot_trajectory_rotation_adr :  POINTER TO ARRAY [0..1000000] OF LREAL;
	
	_robot_fb_motor_1_adr : POINTER TO ARRAY [0..1_000_000] OF LINT;
	_robot_fb_motor_2_adr : POINTER TO ARRAY [0..1_000_000] OF LINT;
	_robot_tg_motor_1_adr : POINTER TO ARRAY [0..1_000_000] OF LINT;
	_robot_tg_motor_2_adr : POINTER TO ARRAY [0..1_000_000] OF LINT;
	
	_robot_trajectory_length: DINT;
	_robot_trajectory_index:DINT;
END_VAR
VAR_STAT
END_VAR
VAR_IN_OUT
END_VAR

IF _robot_interface_adr^.robot_mode=robot_modes_t.CSP AND _robot_interface_adr^.robot_enabled THEN
	CASE _robot_state OF
		robot_traj_states_t.START:
			_motor_pp_scheduler_adr^[0].activate();
			_motor_pp_scheduler_adr^[1].activate();
			InverseKinematics(target_dist:=_robot_trajectory_extension_adr^[0],
							  target_angle:=_robot_trajectory_rotation_adr^[0],
							  motor_axis1_angle=>_target_motor_angles[0],
							  motor_axis2_angle=>_target_motor_angles[1]);
			_motor_pp_scheduler_adr^[0].start_operation(target_position:=_target_motor_angles[0],
				change_immediately:=TRUE, reference_coordinate:=FALSE, push_operation:=FALSE);
			_motor_pp_scheduler_adr^[1].start_operation(target_position:=_target_motor_angles[1],
				change_immediately:=TRUE, reference_coordinate:=FALSE, push_operation:=FALSE);
			_robot_state := robot_traj_states_t.RESET;
		robot_traj_states_t.RESET:
			IF(_motor_pp_scheduler_adr^[0].get_state()=motor_pp_states_t.END AND _motor_pp_scheduler_adr^[1].get_state()=motor_pp_states_t.END) THEN
				_robot_state:=robot_traj_states_t.READY;
			END_IF
		robot_traj_states_t.TRIG:
			_motor_csp_scheduler_adr^[0].activate();
			_motor_csp_scheduler_adr^[1].activate();
			_motor_csp_scheduler_adr^[0].set_position(_target_motor_angles[0]);
			_motor_csp_scheduler_adr^[1].set_position(_target_motor_angles[1]);
			_robot_trajectory_index:=0;
			_robot_state:=robot_traj_states_t.EXEC;
		robot_traj_states_t.EXEC:
			IF(_robot_trajectory_index < _robot_trajectory_length) THEN
				InverseKinematics(	target_dist:=_robot_trajectory_extension_adr^[_robot_trajectory_index],
									target_angle:=_robot_trajectory_rotation_adr^[_robot_trajectory_index],
									motor_axis1_angle=>_target_motor_angles[0],
									motor_axis2_angle=>_target_motor_angles[1]);
				
				_robot_tg_motor_1_adr^[_robot_trajectory_index] := _target_motor_angles[0];
				_robot_tg_motor_2_adr^[_robot_trajectory_index] := _target_motor_angles[1];
				_robot_fb_motor_1_adr^[_robot_trajectory_index] := _motor_interface_adr^[0].feedback_position;
				_robot_fb_motor_2_adr^[_robot_trajectory_index] := _motor_interface_adr^[1].feedback_position;
				_motor_csp_scheduler_adr^[0].set_position(_target_motor_angles[0]);
				_motor_csp_scheduler_adr^[1].set_position(_target_motor_angles[1]);
				_robot_trajectory_index:=_robot_trajectory_index+1;
			ELSE
				_robot_state:=robot_traj_states_t.END;
			END_IF
		robot_traj_states_t.END:
			IF(_robot_trajectory_index < 1_000_000 AND _robot_trajectory_index < _robot_trajectory_length+1000) THEN
				_robot_tg_motor_1_adr^[_robot_trajectory_index] := _target_motor_angles[0];
				_robot_tg_motor_2_adr^[_robot_trajectory_index] := _target_motor_angles[1];
				_robot_fb_motor_1_adr^[_robot_trajectory_index] := _motor_interface_adr^[0].feedback_position;
				_robot_fb_motor_2_adr^[_robot_trajectory_index] := _motor_interface_adr^[1].feedback_position;
				_robot_trajectory_index:=_robot_trajectory_index+1;
			END_IF
	END_CASE
END_IF

{attribute 'TcRpcEnable'}
METHOD activate : BOOL
VAR_INPUT
	
END_VAR
_robot_interface_adr^.robot_mode:=robot_modes_t.CSP;
_robot_state:=robot_traj_states_t.END;
END_METHOD

METHOD FB_init : BOOL
VAR_INPUT
	bInitRetains : BOOL; // if TRUE, the retain variables are initialized (warm start / cold start)
	bInCopyCode : BOOL;  // if TRUE, the instance afterwards gets moved into the copy code (online change)
	robot_interface_adr: POINTER TO RobotInterface;
	robot_trajectory_extension_adr : POINTER TO ARRAY [0..1000000] OF LREAL;
	robot_trajectory_rotation_adr :  POINTER TO ARRAY [0..1000000] OF LREAL;
	robot_fb_motor_1_adr : POINTER TO ARRAY [0..1_000_000] OF LREAL;
	robot_fb_motor_2_adr : POINTER TO ARRAY [0..1_000_000] OF LREAL;
	robot_tg_motor_1_adr : POINTER TO ARRAY [0..1_000_000] OF LREAL;
	robot_tg_motor_2_adr : POINTER TO ARRAY [0..1_000_000] OF LREAL;
END_VAR
_robot_interface_adr:=robot_interface_adr;
_motor_pp_scheduler_adr:=robot_interface_adr^.motor_pp_scheduler_adr;
_motor_hm_scheduler_adr:=robot_interface_adr^.motor_hm_scheduler_adr;
_motor_csp_scheduler_adr:=robot_interface_adr^.motor_csp_scheduler_adr;
_motor_interface_adr:=robot_interface_adr^.motor_interface_adr;
_robot_trajectory_extension_adr := robot_trajectory_extension_adr;
_robot_trajectory_rotation_adr := robot_trajectory_rotation_adr;

	_robot_fb_motor_1_adr := robot_fb_motor_1_adr;
	_robot_fb_motor_2_adr := robot_fb_motor_2_adr;
	_robot_tg_motor_1_adr := robot_tg_motor_1_adr;
	_robot_tg_motor_2_adr := robot_tg_motor_2_adr;
END_METHOD

{attribute 'TcRpcEnable'}
METHOD get_state : robot_traj_states_t
VAR_INPUT
END_VAR
get_state:=_robot_state;
END_METHOD

{attribute 'TcRpcEnable'}
METHOD set_trajectory_length : BOOL
VAR_INPUT
	robot_trajectory_length: DINT;
END_VAR
_robot_trajectory_length:=robot_trajectory_length;
END_METHOD

{attribute 'TcRpcEnable'}
METHOD start_operation : BOOL
VAR_INPUT
END_VAR
_robot_interface_adr^.robot_enabled:=TRUE;
_robot_state:=robot_traj_states_t.START;
_robot_trajectory_index:=0;
END_METHOD

{attribute 'TcRpcEnable'}
METHOD trigger : BOOL
VAR_INPUT
END_VAR
IF(_robot_state<>robot_traj_states_t.READY) THEN
	RETURN;
ELSE
	_robot_state:=robot_traj_states_t.TRIG;
END_IF
END_METHOD

END_FUNCTION_BLOCK

// ---- POUs/RobotControl/RobotKinematics/MATH/ASIND.TcPOU
FUNCTION ASIND : LREAL
VAR_INPUT
	SINVAL:LREAL;
END_VAR
VAR
END_VAR

ASIND:=RAD_TO_DEG(ASIN(SINVAL));

END_FUNCTION
